// TIA Portal V19 export
// export: Created 2024-08-28T07:39:35.3447141Z, ExportSetting WithDefaults, DisplayName Totally Integrated Automation Portal, DisplayVersion V19 Update 2, DisplayName TIA Portal Openness, DisplayVersion V19 Update 2, DisplayName TIA Portal Version Control Interface, DisplayVersion V19, DisplayName TIA Portal Test Suite Advanced, DisplayVersion V19, DisplayName SINAMICS Startdrive Advanced, DisplayVersion V19 SP1, DisplayName SINAMICS Startdrive G130, G150, S120, S150, SINAMICS MV, G220, S200, S210, DisplayVersion V19 SP1, DisplayName SINAMICS Startdrive G110M, G120, G120C, G120D, G120P, G115D, DisplayVersion V19 SP1, DisplayName STEP 7 Professional, DisplayVersion V19 Update 2, DisplayName STEP 7 CFC, DisplayVersion V19, DisplayName STEP 7 Safety, DisplayVersion V19 Update 1, DisplayName WinCC Basic/Comfort/Advanced, DisplayVersion V19 Update 2, DisplayName SIMATIC Visualization Architect, DisplayVersion V19 Update 2, DisplayName WinCC Unified, DisplayVersion V19 Update 2, DisplayName SIMATIC Visualization Architect, DisplayVersion V19 Update 2
FUNCTION "LTU_GetCycleTime" : Void   // FC2, SCL
TITLE = GetCycleTime
{ S7_Optimized_Access := 'TRUE' }
AUTHOR : DT-AGROM
FAMILY : LTU
NAME : EA2i
VERSION : 0.1
// Measure the duration of processes
// stored: AutoNumber true, IsIECCheckEnabled false, SetENOAutomatically false, UDAEnableTagReadback false
   VAR_OUTPUT
      oError : Bool;   // TRUE: An error occurred during the execution of the FC
      oStatus : Word;   // 16#0000 - 16#7FFF: Status of the FB, 16#8000 - 16#FFFF: Error identification
      oCycleTime : Time;
   END_VAR
   VAR_IN_OUT
      ioLastCallTime : DTL;
   END_VAR
   VAR_TEMP
      tDiagnostic : "LTU_DiagnoticUdt";   // Temp diagnostic type to store internal diagnostic data like status and return value of called FCs and system blocks
      tLastTimeCall : DTL;
      tCurrentTimeCall : DTL;
      tCycleTime : Time;
   END_VAR
   VAR CONSTANT
      BLOCK_NAME : String := 'LTU_GetCycleTime';   // Block Name
      STATUS_NO_ERROR : Word := 16#0000;   // NO error - execution finished without errors
      ERR_UNDEFINED_STATE : Word := 16#8600;   // Error: due to an undefined state in state machine
      ERR_IN_BLOCK_OPERATION : Word := 16#8001;   // Error: Wrong operation of the function block
      ERR_PARAMETRIZATION : Word := 16#8200;   // Error: during parameterization
      ERR_PROCESSING_EXTERN : Word := 16#8400;   // Error: when processing from outside (e. g. wrong I/O signals, axis not referenced)
      ERR_PROCESSING_INTERN : Word := 16#8600;   // Error: when processing internally (e. g. when calling a system function)
      ERR_AREA_RESERVED : Word := 16#8800;   // Error: Reserved area
      ERR_USER_DEFINED_CLASSES : Word := 16#9000;   // Error: User-defined error classes
   END_VAR
BEGIN
   REGION BLOCK HEADER
       //=======================================================================================================================================
       // AGROMOUSQUETAIRES _ EA2i // 
       // --------------------------------------------------------------------------------------------------------------------------------------
       // Library: LTU
       // Title : GetCycleTime
       // Function : Measure the duration of processes
       // --------------------------------------------------------------------------------------------------------------------------------------
       // Change tracking :
       // Version      Date            Company                 Author                    Change(s)
       // 00.00.01     14/01/2021      AgroMousquetaires       Thomas Heurtault          Initial version - standard LTU
       //=======================================================================================================================================
   END_REGION
   REGION INITIALISATION
       //  TODO : Use this region for initialize or refresh functionality : tempVariable, diagnostics, etc.
       //         1. Initialized temporary enable state

       #tDiagnostic.status := #STATUS_NO_ERROR;
       #tDiagnostic.subStatus := #STATUS_NO_ERROR;

       #tLastTimeCall := #ioLastCallTime;
       #tCurrentTimeCall := DTL#1970-01-01-0:0:0.0;
       #tCycleTime := T#0ms;

   END_REGION
   REGION FUNCTION
       //  TODO : Use this region for application specific code

       #tDiagnostic.subStatus := INT_TO_WORD(RD_SYS_T(#tCurrentTimeCall));
       #tCycleTime := T_DIFF(IN1 := #tCurrentTimeCall, IN2 := #tLastTimeCall);
       IF T#0ms>#tCycleTime THEN #tCycleTime:= T#0ms; END_IF;

   END_REGION
   REGION OUTPUTS
       //  TODO : Use this region for write new values in outputs
       //         1. Write outputs

       #oError := #tDiagnostic.status.%X15;
       #oStatus := #tDiagnostic.status;
       //#oDiagnostic  := #tDiagnostic;

       #ioLastCallTime := #tCurrentTimeCall;
       #oCycleTime := #tCycleTime;
   END_REGION
END_FUNCTION
